PROGRAM MAIN
VAR
	MC_Power_1: MC_Power;
	MC_MoveAbsolute_1: MC_MoveAbsolute;
	PowerEnable1: BOOL;				//供电使能
	MoveEnable1: BOOL;				//位移使能
	Pos1: LREAL;					//绝对位置
	Vel1: LREAL;					//速度
	PlcTime: LREAL := 0;			//PLC时间
	PlcCycleTicks: LREAL := 0.01;	//PLC运行循环时间 10ms
	status: INT := 0;				//状态转移变量
	Move1Done: BOOL;
END_VAR

PlcTime := PlcTime + PlcCycleTicks;

CASE status OF
	0://初始化
		PowerEnable1 := FALSE;
		MoveEnable1 := FALSE;
		status := 1;
	1://等待3秒，供电&位移使能
		IF PlcTime > 3 THEN
			PowerEnable1 := TRUE;
			MoveEnable1 := TRUE;
			status := 2;
		END_IF
	2://设置移动距离&速度
		Pos1 := 22;
		Vel1 := 1;
		status := 3;
	3://等待移动结束
		IF Move1Done THEN
			status := 4;
		END_IF
	4://
		PowerEnable1 := FALSE;
		MoveEnable1 := FALSE;
END_CASE

ACTION MoveAbsolute:
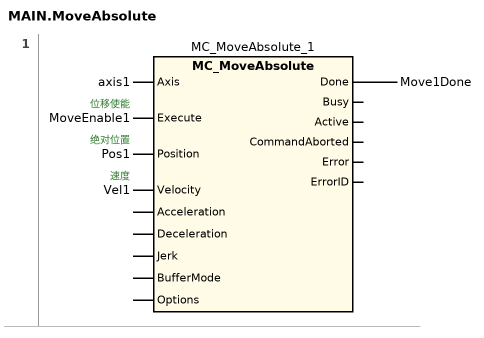
// NETWORK 1
//   MoveEnable1: 位移使能
//   Pos1: 绝对位置
//   Vel1: 速度
MC_MoveAbsolute_1(Axis := axis1, Execute := MoveEnable1, Position := Pos1, Velocity := Vel1); // MC_MoveAbsolute
Move1Done := MC_MoveAbsolute_1.Done;
END_ACTION

ACTION Power:
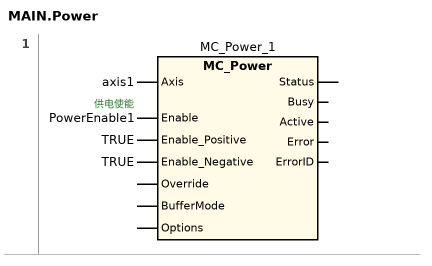
// NETWORK 1
//   PowerEnable1: 供电使能
MC_Power_1(Axis := axis1, Enable := PowerEnable1, Enable_Positive := TRUE, Enable_Negative := TRUE); // MC_Power
END_ACTION

END_PROGRAM

(* stored: Version 1.1.0.1, ProductVersion 3.1.0.38
   POU MAIN: Id {86a9bdf6-f6ba-4ca8-a337-d5afcdfba00d}, SpecialFunc None
   Action MoveAbsolute: Id {7d02e69e-06c7-482e-a944-4db12940c6e4}
   Action Power: Id {bc0a14a0-efeb-4a9c-8cc7-0c3047bb6d6d} *)
